Fanuc KAREL source: ka00185.KL

PROGRAM KA00185
%STACKSIZE=65535
%PRIORITY=65535
%NOLOCKGROUP
VAR
SRC : ARRAY[4] OF BYTE
DST : ARRAY[4] OF BYTE
BEGIN
-- UNRESOLVED_PC line 7 opcodes [22 22 1E] marker_code=0
END KA00185
